{attribute 'linkalways'} 
{attribute 'no_explicit_call' := 'This FB is a CLASS and must be accessed using methods or properties'}
{attribute 'enable_dynamic_creation'}
FUNCTION_BLOCK _ETcVnClusteringAlgorithm EXTENDS EnumDatatypeBase
VAR
	localData : ETcVnClusteringAlgorithm;
	activeData : REFERENCE TO ETcVnClusteringAlgorithm;
	enumBaseDatatype : _DINT(localData);
END_VAR

METHOD PRIVATE AddLocalEnumeration
VAR_INPUT
	Enumeration : T_MAXSTRING;
	Value : ETcVnClusteringAlgorithm;
END_VAR
AddEnumeration(Enumeration, Value);
END_METHOD

PROPERTY PUBLIC Address : PVOID
GET
Address := ADR(activeData);
END_GET
END_PROPERTY

METHOD PUBLIC ClearReference
VAR_INPUT
END_VAR
activeData REF= localData;
SetBaseDatatypeReference();
END_METHOD

METHOD PUBLIC Clone : I_Datatype
VAR
    pClone : POINTER TO _ETcVnClusteringAlgorithm;
END_VAR
pClone := __NEW(_ETcVnClusteringAlgorithm(InitialValue := Value));
Clone := pClone^;
END_METHOD

METHOD FB_init : BOOL
VAR_INPUT
	bInitRetains : BOOL; // if TRUE, the retain variables are initialized (warm start / cold start)
	bInCopyCode : BOOL;  // if TRUE, the instance afterwards gets moved into the copy code (online change)
	InitialValue : ETcVnClusteringAlgorithm;
END_VAR
localData := InitialValue;
AddBaseDatatype(enumBaseDatatype);
ClearReference();

AddLocalEnumeration('TCVN_CA_KMEANSPP', ETcVnClusteringAlgorithm.TCVN_CA_KMEANSPP);
AddLocalEnumeration('TCVN_CA_LBG', ETcVnClusteringAlgorithm.TCVN_CA_LBG);
END_METHOD

PROPERTY PUBLIC Identifier : T_MAXSTRING
GET
Identifier := 'ETcVnClusteringAlgorithm';
END_GET
END_PROPERTY

METHOD IsEnumeratorValueEqual : BOOL
VAR_INPUT
	Enumerator : I_KeyValueForwardEnumerator;
END_VAR
VAR
	storedValue : ETcVnClusteringAlgorithm;
END_VAR
IF NOT Enumerator.TryGet(storedValue) THEN
	RETURN;
END_IF

IsEnumeratorValueEqual := storedValue = activeData;
END_METHOD

METHOD PUBLIC MakeReferenceTo
VAR_INPUT
	ReferenceTarget : REFERENCE TO ETcVnCalibrationPatternOrigin;
END_VAR
activeData REF= ReferenceTarget;
SetBaseDatatypeReference();
END_METHOD

METHOD PROTECTED SetBaseDatatypeReference
VAR_INPUT
END_VAR
enumBaseDatatype.MakeReferenceTo(activeData);
END_METHOD

PROPERTY PUBLIC Size : UDINT
GET
Size := SIZEOF(activeData);
END_GET
END_PROPERTY

METHOD TryMakeReferenceTo : BOOL
VAR_INPUT
	Target : I_Datatype;
END_VAR
VAR
	targetAsEnum : I_EnumDatatype;
	pTargetData : POINTER TO ETcVnClusteringAlgorithm;
END_VAR
IF NOT Target.TryResolveAsEnumDatatype(targetAsEnum) THEN
	RETURN;
END_IF

IF targetAsEnum.Identifier <> Identifier THEN
	RETURN;
END_IF

pTargetData := Target.Address;
activeData REF= pTargetData^;
SetBaseDatatypeReference();
TryMakeReferenceTo := TRUE;
END_METHOD

PROPERTY PUBLIC Value : ETcVnClusteringAlgorithm
GET
Value := activeData;
END_GET
SET
activeData := Value;
END_SET
END_PROPERTY

END_FUNCTION_BLOCK

(* stored: Version 1.1.0.1, ProductVersion 3.1.4024.12
   POU _ETcVnClusteringAlgorithm: Id {276c8f38-e538-44c5-92df-6832fa0ee740}, SpecialFunc None
   Folder Constructor: Id {2750bd5b-925e-4f50-9bbd-f47f1b52f223}
   Folder Private: Id {343b4180-5443-4fdf-82e4-5ea54836fa1e}
   Folder Protected: Id {af4b0071-04d4-4562-b7d7-a62fe10f127b}
   Method AddLocalEnumeration: Id {dcb45ecd-8097-4fc7-9a1c-e113ebb66a58}
   Property Address: Id {898216eb-b0b2-41c0-826e-9413c6712e37}
   Get Get: Id {523666c2-bedd-4fe3-b952-3ff9add4c180}
   Method ClearReference: Id {b1a40e05-b357-40f2-99bb-61f9d5308a8d}
   Method Clone: Id {651dcbd4-1229-43e7-a64b-aacca98bc188}
   Method FB_init: Id {93105a62-b495-409d-b5a7-185cb3c463c9}
   Property Identifier: Id {fd71f75c-89f6-48f9-b415-7fd4863854e7}
   Get Get: Id {1b57410b-5ba0-4cf1-8101-cbfb638fbc5f}
   Method IsEnumeratorValueEqual: Id {1e4ce020-7464-446a-a323-8e2a8702e02c}
   Method MakeReferenceTo: Id {40d6fd12-6339-4332-a859-e95dcd6c11e8}
   Method SetBaseDatatypeReference: Id {ca0f46c8-6542-48a5-b824-910c9ced8afa}
   Property Size: Id {ba473316-556f-4d17-a648-3219f7681f96}
   Get Get: Id {a6ba8a23-8c12-4d8e-a34f-be1a8ebc3427}
   Method TryMakeReferenceTo: Id {ca39e4f5-131b-40a4-89ff-98d4aba524a1}
   Property Value: Id {364101c0-b561-42ec-817e-ef4735290591}
   Get Get: Id {8b3055b2-921b-4462-baec-5116c031defa}
   Set Set: Id {e7693a63-d9e7-41ff-add3-ec707427c854} *)
